FUNCTION_BLOCK WrapMachine
VAR_OUTPUT
	error AT %I* : BOOL;
	ready AT %I* : BOOL;
	busy AT %I* : BOOL;
	done (*AT %I**) : BOOL;
	home AT %I* : BOOL;
	
	rotations AT %Q* : INT;
	execute AT %Q* : BOOL;
	enable AT %Q* : BOOL;
	reset AT %Q* : BOOL;
	
	timeout : BOOL;
END_VAR
VAR
	holdPost : TON;
	delay : TON;
	
	start : BOOL;
	step : (SETUP, RUN, WAIT);
END_VAR
VAR_STAT CONSTANT
	pulseTime : TIME := T#100MS;
	holdTime : TIME := T#500MS;
	maxDelay : TIME := T#30S;
END_VAR

holdPost(IN:= , PT:= holdTime, Q=> , ET=> );
delay(IN:= step > 0, PT:= maxDelay, Q=> , ET=> );

IF delay.Q THEN
	delay.IN := FALSE;
	timeout := TRUE;
	busy := FALSE;
	step := SETUP;
END_IF

CASE step OF
	SETUP:
		busy := FALSE;
		IF error THEN
			reset := NOT reset;
			enable := FALSE;//NOT enable;
			
		ELSE
			reset := FALSE;
			enable := TRUE;
			
			IF start THEN
				start := FALSE;
				step := RUN;
			END_IF
			
		END_IF
	
	RUN:
		execute := TRUE;
		IF execute AND NOT home THEN
			execute := FALSE;
			step := WAIT;
		END_IF
		
	WAIT:
		IF home THEN
			holdPost.IN := TRUE;
			enable := FALSE;
			execute := FALSE;
		END_IF
		
		IF holdPost.Q THEN
			holdPost.IN := FALSE;
			done := TRUE;
			step := 0;
		END_IF
		
END_CASE

METHOD clear : BOOL
VAR_INPUT
END_VAR
(*
reset should be continuously called until machine returns evidence that it is ready again
machine is expected to not respond to reset signals if it is already in an idle state
*)
enable := FALSE;
execute := FALSE;

IF error THEN
	reset := NOT reset;
	clear := NOT error;

ELSE
	reset := FALSE;
	clear := TRUE;
	
END_IF
END_METHOD

METHOD wrap : BOOL
VAR_INPUT
	reqRotations : INT;
END_VAR
IF ready AND NOT busy AND NOT error THEN
	rotations := reqRotations;
	busy := TRUE;
	start := TRUE;
	wrap := TRUE;
END_IF
END_METHOD

END_FUNCTION_BLOCK

(* stored: Version 1.1.0.1, ProductVersion 3.1.4024.11
   POU WrapMachine: Id {a3ca7ffd-0355-457d-b5e4-e9e36ee78e64}, SpecialFunc None
   Method clear: Id {809335de-2787-442d-8a0b-81b9b3831244}
   Method wrap: Id {1ec79807-3015-428d-b6b1-6b5d17802bae} *)
